Yaskawa INFORM job: A-5-08279-80-0-M.JBI

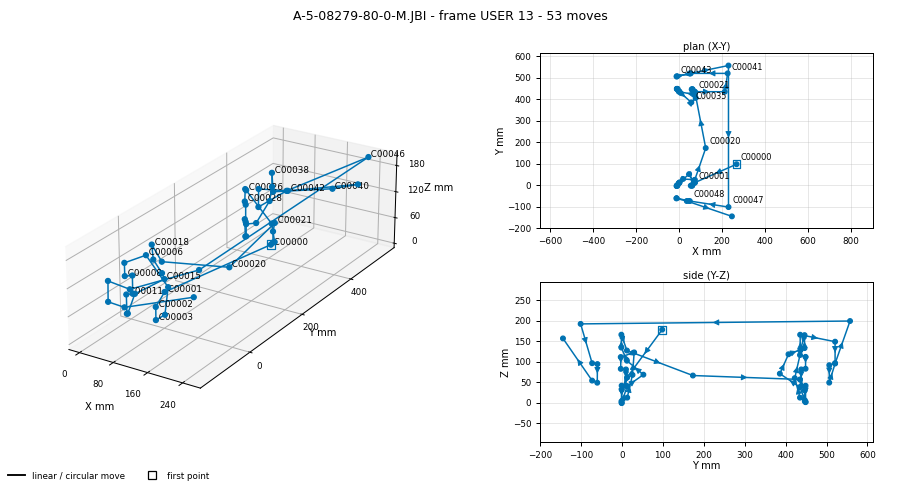
[picture p0: tool path of A-5-08279-80-0-M.JBI in frame USER 13, 53 of 53 moves have a stored position in this frame; points joined in program order, loops and branches not executed]
/JOB
//NAME A-5-08279-80-0-M
///FOLDERNAME PART_420-08279-80
//POS
///NPOS 53,0,53,0,0,0
///USER 13
///TOOL 4
///POSTYPE USER
///RECTAN
///RCONF 1,0,0,0,0,0,0,0,0,0,0,0,0,0,0,0,0,0,0,0,0,0,0,0
C00000=267.003,98.367,178.621,-96.7910,26.0612,130.3914
C00001=73.206,12.887,62.532,-108.1130,33.6440,124.7280
C00002=60.671,-0.651,32.061,-108.1124,33.6411,124.7298
C00003=60.874,-1.212,3.334,-108.1142,33.6462,124.7273
C00004=73.207,12.886,12.496,-108.1130,33.6440,124.7280
C00005=73.209,25.753,68.034,-108.1130,33.6440,124.7280
C00006=18.285,29.861,123.023,-105.1660,8.3780,132.7380
C00007=-11.539,-2.869,111.733,-105.6879,27.7518,134.0459
C00008=-11.243,-2.886,82.832,-105.6905,27.7500,134.0449
C00009=-1.744,9.833,81.413,-106.8820,26.9670,127.1640
C00010=-1.744,9.833,41.151,-106.8820,26.9670,127.1640
C00011=-10.039,-0.764,41.755,-105.8464,28.0438,133.0351
C00012=-9.761,-0.631,-0.899,-124.6798,17.6320,128.8675
C00013=-7.562,-0.629,0.044,-124.6779,17.6312,128.8671
C00014=1.309,12.886,40.637,-115.9500,15.0640,123.8880
C00015=46.568,52.366,68.637,-115.9500,15.0640,123.8880
C00016=68.126,12.203,102.713,-51.9240,65.1860,170.4170
C00017=57.254,-1.496,134.820,-51.9224,65.1860,170.4182
C00018=54.145,-1.424,166.316,-51.9156,65.1891,170.4218
C00019=68.127,12.203,127.579,-51.9240,65.1860,170.4170
C00020=123.702,173.377,66.504,-51.9240,65.1860,170.4170
C00021=73.207,435.046,56.988,108.1130,33.6440,-124.7280
C00022=61.863,446.758,30.241,108.1130,33.6439,-124.7276
C00023=62.002,446.808,4.162,108.1113,33.6487,-124.7260
C00024=73.207,435.046,12.497,108.1130,33.6440,-124.7280
C00025=73.208,422.239,60.087,108.1130,33.6440,-124.7280
C00026=1.310,435.046,116.590,106.4700,24.0930,-128.1180
C00027=-9.553,448.700,112.134,105.5211,25.1069,-133.5885
C00028=-10.606,448.654,83.063,105.5185,25.1075,-133.5880
C00029=-1.744,438.100,81.414,106.4700,24.0930,-128.1180
C00030=-1.744,438.100,41.152,106.4700,24.0930,-128.1180
C00031=-10.576,448.703,41.619,105.1161,25.4804,-135.7639
C00032=-9.077,448.650,1.453,122.7053,28.9561,-128.7016
C00033=-6.926,448.642,2.115,122.7040,28.9586,-128.6998
C00034=1.310,435.046,37.856,114.8060,13.4990,-125.4170
C00035=56.824,385.802,71.014,114.8060,13.4990,-125.4170
C00036=76.829,406.941,118.422,51.9240,65.1860,-170.4170
C00037=59.248,446.146,133.508,51.9214,65.1887,-170.4176
C00038=58.580,446.196,165.210,51.9245,65.1880,-170.4161
C00039=68.127,435.729,127.579,51.9240,65.1860,-170.4170
C00040=212.373,435.445,166.233,51.9240,65.1860,-170.4170
C00041=225.757,520.809,149.229,-64.9600,52.3020,155.2860
C00042=54.000,520.810,96.661,-64.9600,52.3020,155.2860
C00043=-11.222,506.636,91.772,-64.9639,52.3006,155.2847
C00044=-11.590,506.512,49.143,-64.9609,52.3037,155.2848
C00045=50.732,520.809,95.877,-64.9600,52.3020,155.2860
C00046=229.531,557.327,199.687,42.3120,70.9810,-117.7980
C00047=229.653,-100.956,192.660,69.2460,43.0800,-149.5110
C00048=49.647,-72.877,96.659,69.2460,43.0800,-149.5110
C00049=-11.715,-59.900,94.479,69.2464,43.0793,-149.5107
C00050=-12.366,-60.325,48.967,69.2475,43.0789,-149.5111
C00051=35.736,-72.877,54.138,69.2460,43.0800,-149.5110
C00052=245.487,-144.122,157.206,69.2470,43.0790,-149.5110
///TOOL 0
///POSTYPE ANGLE
///ANGLE
EC00000=15.0000
///TOOL 4
EC00001=15.0000
///TOOL 0
EC00002=15.0000
EC00003=15.0000
///TOOL 4
EC00004=15.0000
EC00005=15.0000
EC00006=15.0000
///TOOL 0
EC00007=15.0000
EC00008=15.0000
///TOOL 4
EC00009=15.0000
EC00010=15.0000
///TOOL 0
EC00011=15.0000
EC00012=14.9994
EC00013=14.9994
///TOOL 4
EC00014=15.0000
EC00015=15.0000
EC00016=15.0000
///TOOL 0
EC00017=15.0000
EC00018=15.0000
///TOOL 4
EC00019=15.0000
EC00020=15.0000
EC00021=15.0000
///TOOL 0
EC00022=15.0000
EC00023=15.0000
///TOOL 4
EC00024=15.0000
EC00025=15.0000
EC00026=15.0000
///TOOL 0
EC00027=15.0000
EC00028=15.0000
///TOOL 4
EC00029=15.0000
EC00030=15.0000
///TOOL 0
EC00031=15.0000
EC00032=15.0000
EC00033=15.0000
///TOOL 4
EC00034=15.0000
EC00035=15.0000
EC00036=15.0000
///TOOL 0
EC00037=15.0000
EC00038=15.0000
///TOOL 4
EC00039=15.0000
EC00040=15.0000
EC00041=15.0000
EC00042=15.0000
///TOOL 0
EC00043=15.0000
EC00044=15.0000
///TOOL 4
EC00045=15.0000
EC00046=15.0000
EC00047=15.0000
EC00048=15.0000
///TOOL 0
EC00049=15.0000
EC00050=15.0000
///TOOL 4
EC00051=15.0000
EC00052=15.0000
//INST
///DATE 2021/10/29 11:36
///ATTR SC,RW,RJ
////FRAME USER 13
///GROUP1 RB1
///GROUP2 ST2
NOP
'Path Start: PP56
MOVJ C00000 VJ=100.00  +MOVJ EC00000
SMOVL C00001 V=1250.0  +MOVJ EC00001
SMOVL C00002 V=300.0  +MOVJ EC00002
ARCON ASF#(953)
SMOVL C00003 V=8.5  +MOVJ EC00003
ARCOF AEF#(953)
SMOVL C00004 V=1250.0  +MOVJ EC00004
SMOVL C00005 V=1250.0  +MOVJ EC00005
'Path End
'Path Start: PP54
SMOVL C00006 V=1250.0  +MOVJ EC00006
SMOVL C00007 V=300.0  +MOVJ EC00007
ARCON ASF#(952)
SMOVL C00008 V=6.3  +MOVJ EC00008
ARCOF AEF#(954)
SMOVL C00009 V=300.0  +MOVJ EC00009
SMOVL C00010 V=300.0  +MOVJ EC00010
SMOVL C00011 V=300.0  +MOVJ EC00011
ARCON ASF#(952)
SMOVL C00012 V=6.3  +MOVJ EC00012
SMOVL C00013 V=6.3  +MOVJ EC00013
ARCOF AEF#(954)
SMOVL C00014 V=1250.0  +MOVJ EC00014
SMOVL C00015 V=1250.0  +MOVJ EC00015
'Path End
'Path Start: Path_5
SMOVL C00016 V=1250.0  +MOVJ EC00016
SMOVL C00017 V=1250.0  +MOVJ EC00017
ARCON ASF#(951)
SMOVL C00018 V=8.5  +MOVJ EC00018
ARCOF AEF#(951)
SMOVL C00019 V=1250.0  +MOVJ EC00019
SMOVL C00020 V=1250.0  +MOVJ EC00020
'Path End
'Path Start: PP55
SMOVL C00021 V=1250.0  +MOVJ EC00021
SMOVL C00022 V=300.0  +MOVJ EC00022
ARCON ASF#(953)
SMOVL C00023 V=8.5  +MOVJ EC00023
ARCOF AEF#(953)
SMOVL C00024 V=1250.0  +MOVJ EC00024
SMOVL C00025 V=1250.0  +MOVJ EC00025
'Path End
'Path Start: PP58
SMOVL C00026 V=1250.0  +MOVJ EC00026
SMOVL C00027 V=300.0  +MOVJ EC00027
ARCON ASF#(952)
SMOVL C00028 V=6.3  +MOVJ EC00028
ARCOF AEF#(954)
SMOVL C00029 V=300.0  +MOVJ EC00029
SMOVL C00030 V=300.0  +MOVJ EC00030
SMOVL C00031 V=300.0  +MOVJ EC00031
ARCON ASF#(952)
SMOVL C00032 V=6.3  +MOVJ EC00032
SMOVL C00033 V=6.3  +MOVJ EC00033
ARCOF AEF#(954)
SMOVL C00034 V=1250.0  +MOVJ EC00034
SMOVL C00035 V=1250.0  +MOVJ EC00035
'Path End
'Path Start: Path_4
SMOVL C00036 V=1250.0  +MOVJ EC00036
SMOVL C00037 V=1250.0  +MOVJ EC00037
ARCON ASF#(951)
SMOVL C00038 V=8.5  +MOVJ EC00038
ARCOF AEF#(951)
SMOVL C00039 V=1250.0  +MOVJ EC00039
SMOVL C00040 V=1250.0  +MOVJ EC00040
'Path End
'Path Start: PP57
SMOVL C00041 V=1250.0  +MOVJ EC00041
SMOVL C00042 V=1250.0  +MOVJ EC00042
SMOVL C00043 V=300.0  +MOVJ EC00043
ARCON ASF#(953)
SMOVL C00044 V=8.5  +MOVJ EC00044
ARCOF AEF#(953)
SMOVL C00045 V=1250.0  +MOVJ EC00045
SMOVL C00046 V=1250.0  +MOVJ EC00046
'Path End
'Path Start: PP53
SMOVL C00047 V=1250.0  +MOVJ EC00047
SMOVL C00048 V=1250.0  +MOVJ EC00048
SMOVL C00049 V=300.0  +MOVJ EC00049
ARCON ASF#(953)
SMOVL C00050 V=8.5  +MOVJ EC00050
ARCOF AEF#(953)
SMOVL C00051 V=1250.0  +MOVJ EC00051
SMOVL C00052 V=1250.0  +MOVJ EC00052
'Path End
END
